FUNCTION fnCnvToTarg : T_Arg
VAR_INPUT
	param1:ANY;
END_VAR
VAR
END_VAR


CASE 	 param1.TypeClass OF	
	 __SYSTEM.TYPE_CLASS.TYPE_REAL:
			 fnCnvToTarg.eType	:= E_ArgType.ARGTYPE_REAL;
	 __SYSTEM.TYPE_CLASS.TYPE_INT:
			 fnCnvToTarg.eType	:= E_ArgType.ARGTYPE_INT;	 
	 __SYSTEM.TYPE_CLASS.TYPE_LREAL:
			 fnCnvToTarg.eType	:= E_ArgType.ARGTYPE_LREAL;
	 __SYSTEM.TYPE_CLASS.TYPE_SINT:
			 fnCnvToTarg.eType	:= E_ArgType.ARGTYPE_SINT;	 		
	 __SYSTEM.TYPE_CLASS.TYPE_DINT:
			 fnCnvToTarg.eType	:= E_ArgType.ARGTYPE_DINT;
	 __SYSTEM.TYPE_CLASS.TYPE_USINT:
			 fnCnvToTarg.eType	:= E_ArgType.ARGTYPE_USINT;	 
	 __SYSTEM.TYPE_CLASS.TYPE_UINT:
			 fnCnvToTarg.eType	:= E_ArgType.ARGTYPE_UINT;
	 __SYSTEM.TYPE_CLASS.TYPE_UDINT:
			 fnCnvToTarg.eType	:= E_ArgType.ARGTYPE_UDINT;	 	
	 __SYSTEM.TYPE_CLASS.TYPE_ULINT:
			 fnCnvToTarg.eType	:= E_ArgType.ARGTYPE_ULARGE;
	__SYSTEM.TYPE_CLASS.TYPE_LINT:
			 fnCnvToTarg.eType	:= E_ArgType.ARGTYPE_LARGE;	 			 
	 __SYSTEM.TYPE_CLASS.TYPE_STRING:
			 fnCnvToTarg.eType	:= E_ArgType.ARGTYPE_STRING;
	 __SYSTEM.TYPE_CLASS.TYPE_BOOL:
			 fnCnvToTarg.eType	:= E_ArgType.ARGTYPE_BYTE;//Not a Bug use to convert bool to byte for string format	 
	 __SYSTEM.TYPE_CLASS.TYPE_BYTE:
			 fnCnvToTarg.eType	:= E_ArgType.ARGTYPE_BYTE;
	 __SYSTEM.TYPE_CLASS.TYPE_WORD:
			 fnCnvToTarg.eType	:= E_ArgType.ARGTYPE_WORD;	 		
	 __SYSTEM.TYPE_CLASS.TYPE_DWORD:
			 fnCnvToTarg.eType	:= E_ArgType.ARGTYPE_DWORD;
	 __SYSTEM.TYPE_CLASS.TYPE_ENUM:
	 		IF param1.diSize = SIZEOF(INT) THEN
			 	fnCnvToTarg.eType	:= E_ArgType.ARGTYPE_INT;	
			ELSIF param1.diSize = SIZEOF(DINT) THEN		 
				fnCnvToTarg.eType	:= E_ArgType.ARGTYPE_DINT;	
			ELSIF param1.diSize = SIZEOF(UDINT) THEN		 
				fnCnvToTarg.eType	:= E_ArgType.ARGTYPE_UDINT;			
			ELSIF param1.diSize = SIZEOF(UINT) THEN		 
				fnCnvToTarg.eType	:= E_ArgType.ARGTYPE_UINT;	
			END_IF	
ELSE
	RETURN; 
END_CASE

fnCnvToTarg.pData := param1.pValue;
fnCnvToTarg.cbLen := DINT_TO_UDINT(param1.diSize);

END_FUNCTION

(* stored: Version 1.1.0.1, ProductVersion 3.1.4024.3
   POU fnCnvToTarg: Id {02762320-3576-4a8a-96db-062f502db6f8}, SpecialFunc None *)
